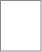
VISUALIZATION V_RolGrp  // 42x52
VAR_IN_OUT
	m_Input_fbRolloGruppe : FB_RolloGruppe;
END_VAR
    Polygon (40,20), colour toggle: (m_Input_fbRolloGruppe.tonRolloAb.Q =0) <> 0, invisible if: (m_Input_fbRolloGruppe.QbOutRolloAb =1) <> 0
    Polygon (40,30), colour toggle: (m_Input_fbRolloGruppe.tonRolloAb.Q =0) <> 0, invisible if: (m_Input_fbRolloGruppe.QbOutRolloAb =0) <> 0
    Polygon (40,20), colour toggle: (m_Input_fbRolloGruppe.bInVisuAuf) <> 0
        tap m_Input_fbRolloGruppe.bInVisuAuf
    Polygon (20,50), colour toggle: (m_Input_fbRolloGruppe.bInVisuAb) <> 0
        tap m_Input_fbRolloGruppe.bInVisuAb
END_VISUALIZATION

(* stored: Version 1.1.0.1, ProductVersion 3.1.4018.10
   Visu V_RolGrp: Id {3cb24806-9534-4c1d-8344-9c44d4b78958} *)
